# B&R Automation Studio project NAELD004C00R10L518F00 (part 31)

#### Local.var - Do Not Change!!!
```iecst
(*2019-06-17*)
(**)
(*Local Action, State & Status*)
VAR
	eAct : eConvAction := ConvActIdle;
	eStat : eConvAction := ConvActIdle;
	eStatus : eFBStatus := Idle;
	udiStatus : UDINT := 0;
	sStatTxt : STRING[200] := '';
	a_sStatText : ARRAY[0..60] OF STRING[200] := ['Idling','Initializing','Initializing With Reverse','Initializing With Pusher','Initializing With Puller','Initializing With Motorised Puller','Initializing With Reject','Initializing With Inspection','Entering Board','Entering Board Until Inlet Signal Off','Entering Board With Reverse','Reversing Board','Reversing Board With Immediate Start Conv','Entering Board With Puller','Entering Board With Reject','Entering Board With Inspection','Pre Exiting Board','Resuming Reject Board',2('Exiting Board'),2('Exiting Board With Pusher'),'Pusher Setting All Control','Pusher Resetting All Control','Pusher Setting Extend','Pusher Setting Retract','Pusher Extending','Pusher Retracting','Puller Setting All Control','Puller Resetting All Control','Puller Setting Extend','Puller Setting Retract','Puller Extending','Puller Retracting','Rotating Setting All Control','Rotating Resetting All Control','Rotating Setting Home','Rotating Setting Remote','Rotating Turning Home','Rotating Turning Remote','Reject Setting All Control','Reject Resetting All Control','Reject Setting Up','Reject Setting Down','Reject Going Up','Reject Going Down','Stopping','Stopping With Pusher','Stopping With Puller','Stopping With Reject','Turning On Motor Signal','Turning On Motor Direction','Turning Off Motor Signal','Turning Off Motor Direction','Turning On All Motor Output','Turning Off All Motor Output',5('')];
END_VAR
(**)
(*Local Alarm*)
VAR
	tyAlmData : tyAlmDat;
	a_tyAlmText : ARRAY[10000..10199] OF tyAlmTxt := [(sAlmText:='Multi Board Detected While Conveyor Initial',sRcyText:='Operation Interrupted By Multiple Board. Remove Extra Boards And Resume Operation.'),(sAlmText:='Board Not Present At Outlet Sensor (L - R) While Conveyor Initial',sRcyText:='Operation Interrupted By Jam Board. Remove The Jam Board To Resume Operation.'),(sAlmText:='Board Not Present At Outlet Sensor (R - L) While Conveyor Initial',sRcyText:='Operation Interrupted By Jam Board. Remove The Jam Board To Resume Operation.'),(sAlmText:='Multi Board Detected While Conveyor Initial With Reverse',sRcyText:='Operation Interrupted By Multiple Board. Remove Extra Boards And Resume Operation.'),(sAlmText:='Board Not Present At Outlet Sensor (L - R) While Conveyor Initial With Reverse',sRcyText:='Operation Interrupted By Jam Board. Remove The Jam Board To Resume Operation.'),(sAlmText:='Board Not Present At Outlet Sensor (R - L) While Conveyor Initial With Reverse',sRcyText:='Operation Interrupted By Jam Board. Remove The Jam Board To Resume Operation.'),(sAlmText:='Pusher Extend Sensor Off Time Out In Retract Check While Conveyor Initial With Pusher',sRcyText:='Sensor Timeout Expired Before Operation Completed. Sensor Operation Is Abnormal. Solve The Error To Resume Operation.'),(sAlmText:='Pusher Retract Sensor On Time Out In Retract Check While Conveyor Initial With Pusher',sRcyText:='Sensor Timeout Expired Before Operation Completed. Sensor Operation Is Abnormal. Solve The Error To Resume Operation.'),(sAlmText:='Pusher Retract Safety Sensor Error In Retract Check While Conveyor Initial With Pusher',sRcyText:='Safety System Has Been Triggered. All Operations Are Disable. Remove the Obstacle That Triggered The Safety Interlock To Resume Operation.'),(sAlmText:='Multi Board Detected While Conveyor Initial With Pusher',sRcyText:='Operation Interrupted By Multiple Board. Remove Extra Boards And Resume Operation.'),(sAlmText:='Board Not Present At Outlet Sensor (L - R) While Conveyor Initial With Pusher',sRcyText:='Operation Interrupted By Jam Board. Remove The Jam Board To Resume Operation.'),(sAlmText:='Board Not Present At Outlet Sensor (R - L) While Conveyor Initial With Pusher',sRcyText:='Operation Interrupted By Jam Board. Remove The Jam Board To Resume Operation.'),(sAlmText:='Rotator Home Sensor On Time Out In Home Check While Conveyor Initial With Puller',sRcyText:='Sensor Timeout Expired Before Operation Completed. Sensor Operation Is Abnormal. Solve The Error To Resume Operation.'),(sAlmText:='Rotator Remote Sensor Off Time Out In Home Check While Conveyor Initial With Puller',sRcyText:='Sensor Timeout Expired Before Operation Completed. Sensor Operation Is Abnormal. Solve The Error To Resume Operation.'),(sAlmText:='Rotator Home Safety Sensor Error In Home Check While Conveyor Initial With Puller',sRcyText:='Safety System Has Been Triggered. All Operations Are Disable. Remove the Obstacle That Triggered The Safety Interlock To Resume Operation.'),(sAlmText:='Puller Extend Sensor Off Time Out In Retract Check While Conveyor Initial With Puller',sRcyText:='Sensor Timeout Expired Before Operation Completed. Sensor Operation Is Abnormal. Solve The Error To Resume Operation.'),(sAlmText:='Puller Retract Sensor On Time Out In Retract Check While Conveyor Initial With Puller',sRcyText:='Sensor Timeout Expired Before Operation Completed. Sensor Operation Is Abnormal. Solve The Error To Resume Operation.'),(sAlmText:='Puller Retract Safety Sensor Error In Retract Check While Conveyor Initial With Puller',sRcyText:='Safety System Has Been Triggered. All Operations Are Disable. Remove the Obstacle That Triggered The Safety Interlock To Resume Operation.'),(sAlmText:='Multi Board Detected While Conveyor Initial With Puller',sRcyText:='Operation Interrupted By Multiple Board. Remove Extra Boards And Resume Operation.'),(sAlmText:='Board Not Present At Outlet Sensor (L - R) While Conveyor Initial With Puller',sRcyText:='Operation Interrupted By Jam Board. Remove The Jam Board To Resume Operation.'),(sAlmText:='Board Not Present At Outlet Sensor (R - L) While Conveyor Initial With Puller',sRcyText:='Operation Interrupted By Jam Board. Remove The Jam Board To Resume Operation.'),(sAlmText:='Multi Board Detected While Conveyor Enter Board',sRcyText:='Operation Interrupted By Multiple Board. Remove Extra Boards And Resume Operation.'),(sAlmText:='Multi Board Detected While Conveyor Enter Board With Reverse',sRcyText:='Operation Interrupted By Multiple Board. Remove Extra Boards And Resume Operation.'),(sAlmText:='Puller Extend Sensor On Time Out In Extend Check While Conveyor Enter With Puller',sRcyText:='Sensor Timeout Expired Before Operation Completed. Sensor Operation Is Abnormal. Solve The Error To Resume Operation.'),(sAlmText:='Puller Retract Sensor Off Time Out In Extend Check While Conveyor Enter With Puller',sRcyText:='Sensor Timeout Expired Before Operation Completed. Sensor Operation Is Abnormal. Solve The Error To Resume Operation.'),(sAlmText:='Puller Extend Safety Sensor Error In Extend Check While Conveyor Enter With Puller',sRcyText:='Safety System Has Been Triggered. All Operations Are Disable. Remove the Obstacle That Triggered The Safety Interlock To Resume Operation.'),(sAlmText:='Rotator Home Sensor Off Time Out In Remote Check While Conveyor Enter With Puller',sRcyText:='Sensor Timeout Expired Before Operation Completed. Sensor Operation Is Abnormal. Solve The Error To Resume Operation.'),(sAlmText:='Rotator Remote Sensor On Time Out In Remote Check While Conveyor Enter With Puller',sRcyText:='Sensor Timeout Expired Before Operation Completed. Sensor Operation Is Abnormal. Solve The Error To Resume Operation.'),(sAlmText:='Rotator Remote Safety Sensor Error In Remote Check While Conveyor Enter With Puller',sRcyText:='Safety System Has Been Triggered. All Operations Are Disable. Remove the Obstacle That Triggered The Safety Interlock To Resume Operation.'),(sAlmText:='Puller Extend Sensor Off Time Out In Retract Check While Conveyor Enter With Puller',sRcyText:='Sensor Timeout Expired Before Operation Completed. Sensor Operation Is Abnormal. Solve The Error To Resume Operation.'),(sAlmText:='Puller Retract Sensor On Time Out In Retract Check While Conveyor Enter With Puller',sRcyText:='Sensor Timeout Expired Before Operation Completed. Sensor Operation Is Abnormal. Solve The Error To Resume Operation.'),(sAlmText:='Puller Retract Safety Sensor Error In Retract Check While Conveyor Enter With Puller',sRcyText:='Safety System Has Been Triggered. All Operations Are Disable. Remove the Obstacle That Triggered The Safety Interlock To Resume Operation.'),(sAlmText:='Rotator Home Sensor On Time Out In Home Check While Conveyor Enter With Puller',sRcyText:='Sensor Timeout Expired Before Operation Completed. Sensor Operation Is Abnormal. Solve The Error To Resume Operation.'),(sAlmText:='Rotator Remote Sensor Off Time Out In Home Check While Conveyor Enter With Puller',sRcyText:='Sensor Timeout Expired Before Operation Completed. Sensor Operation Is Abnormal. Solve The Error To Resume Operation.'),(sAlmText:='Rotator Home Safety Sensor Error In Home Check While Conveyor Enter With Puller',sRcyText:='Safety System Has Been Triggered. All Operations Are Disable. Remove the Obstacle That Triggered The Safety Interlock To Resume Operation.'),(sAlmText:='Multi Board Detected While Conveyor Enter With Puller',sRcyText:='Operation Interrupted By Multiple Board. Remove Extra Boards And Resume Operation.'),(sAlmText:='Multi Board Detected While Conveyor Pre-Exit Board',sRcyText:='Operation Interrupted By Multiple Board. Remove Extra Boards And Resume Operation.'),(sAlmText:='Board Missing While Conveyor Pre-Exit Board',sRcyText:='Operation Interrupted By Jam Board. Remove The Jam Board To Resume Operation.'),(sAlmText:='Multi Board Detected While Conveyor Exit Board',sRcyText:='Operation Interrupted By Multiple Board. Remove Extra Boards And Resume Operation.'),(sAlmText:='Multi Board Detected While Conveyor Exit Board With Pusher',sRcyText:='Operation Interrupted By Multiple Board. Remove Extra Boards And Resume Operation.'),(sAlmText:='Pusher Extend Sensor On Time Out In Extend Check While Conveyor Exit Board With Pusher',sRcyText:='Sensor Timeout Expired Before Operation Completed. Sensor Operation Is Abnormal. Solve The Error To Resume Operation.'),(sAlmText:='Pusher Retract Sensor Off Time Out In Extend Check While Conveyor Exit Board With Pusher',sRcyText:='Sensor Timeout Expired Before Operation Completed. Sensor Operation Is Abnormal. Solve The Error To Resume Operation.'),(sAlmText:='Pusher Extend Safety Sensor Error In Extend Check While Conveyor Exit Board With Pusher',sRcyText:='Safety System Has Been Triggered. All Operations Are Disable. Remove the Obstacle That Triggered The Safety Interlock To Resume Operation.'),(sAlmText:='Pusher Extend Sensor Off Time Out In Retract Check While Conveyor Exit Board With Pusher',sRcyText:='Sensor Timeout Expired Before Operation Completed. Sensor Operation Is Abnormal.Solve The Error To Resume Operation.'),(sAlmText:='Pusher Retract Sensor On Timeout In Retract Check While Conveyor Exit Board With Pusher',sRcyText:='Sensor Timeout Expired Before Operation Completed. Sensor Operation Is Abnormal. Solve The Error To Resume Operation.'),(sAlmText:='Pusher Retract Safety Sensor Error In Retract Check While Conveyor Exit Board With Pusher',sRcyText:='Safety System Has Been Triggered. All Operations Are Disable. Remove the Obstacle That Triggered The Safety Interlock To Resume Operation.'),(sAlmText:='Pusher Extend Sensor On Time Out In Extend Check While Pusher Extend',sRcyText:='Sensor Timeout Expired Before Operation Completed. Sensor Operation Is Abnormal. Solve The Error To Resume Operation.'),(sAlmText:='Pusher Retract Sensor Off Time Out In Extend Check While Pusher Extend',sRcyText:='Sensor Timeout Expired Before Operation Completed. Sensor Operation Is Abnormal. Solve The Error To Resume Operation.'),(sAlmText:='Pusher Extend Safety Sensor Error In Extend Check While Pusher Extend',sRcyText:='Safety System Has Been Triggered. All Operations Are Disable. Remove the Obstacle That Triggered The Safety Interlock To Resume Operation.'),(sAlmText:='Pusher Extend Sensor Off Time Out In Retract Check While Pusher Retract',sRcyText:='Sensor Timeout Expired Before Operation Completed. Sensor Operation Is Abnormal. Solve The Error To Resume Operation.'),(sAlmText:='Pusher Retract Sensor On Time Out In Retract Check While Pusher Retract',sRcyText:='Sensor Timeout Expired Before Operation Completed. Sensor Operation Is Abnormal. Solve The Error To Resume Operation.'),(sAlmText:='Pusher Retract Safety Sensor Error In Retract Check While Pusher Retract',sRcyText:='Safety System Has Been Triggered. All Operations Are Disable. Remove the Obstacle That Triggered The Safety Interlock To Resume Operation.'),(sAlmText:='Puller Extend Sensor On Time Out In Extend Check While Puller Extend',sRcyText:='Sensor Timeout Expired Before Operation Completed. Sensor Operation Is Abnormal. Solve The Error To Resume Operation.'),(sAlmText:='Puller Retract Sensor Off Time Out In Extend Check While Puller Extend',sRcyText:='Sensor Timeout Expired Before Operation Completed. Sensor Operation Is Abnormal. Solve The Error To Resume Operation.'),(sAlmText:='Puller Extend Safety Sensor Error In Extend Check While Puller Extend',sRcyText:='Safety System Has Been Triggered. All Operations Are Disable. Remove the Obstacle That Triggered The Safety Interlock To Resume Operation.'),(sAlmText:='Puller Extend Sensor Off Time Out In Retract Check While Puller Retract',sRcyText:='Sensor Timeout Expired Before Operation Completed. Sensor Operation Is Abnormal. Solve The Error To Resume Operation.'),(sAlmText:='Puller Retract Sensor On Time Out In Retract Check While Puller Retract',sRcyText:='Sensor Timeout Expired Before Operation Completed. Sensor Operation Is Abnormal. Solve The Error To Resume Operation.'),(sAlmText:='Puller Retract Safety Sensor Error In Retract Check While Puller Retract',sRcyText:='Safety System Has Been Triggered. All Operations Are Disable. Remove the Obstacle That Triggered The Safety Interlock To Resume Operation.'),(sAlmText:='Rotator Home Sensor On Time Out In Home Check While Rotator Home',sRcyText:='Sensor Timeout Expired Before Operation Completed. Sensor Operation Is Abnormal. Solve The Error To Resume Operation.'),(sAlmText:='Rotator Remote Sensor Off Time Out In Home Check While Rotator Home',sRcyText:='Sensor Timeout Expired Before Operation Completed. Sensor Operation Is Abnormal. Solve The Error To Resume Operation.'),(sAlmText:='Rotator Home Safety Sensor Error In Home Check While Rotator Home',sRcyText:='Safety System Has Been Triggered. All Operations Are Disable. Remove the Obstacle That Triggered The Safety Interlock To Resume Operation.'),(sAlmText:='Rotator Home Sensor Off Time Out In Remote Check While Rotator Remote',sRcyText:='Sensor Timeout Expired Before Operation Completed. Sensor Operation Is Abnormal. Solve The Error To Resume Operation.'),(sAlmText:='Rotator Remote Sensor On Time Out In Remote Check While Rotator Remote',sRcyText:='Sensor Timeout Expired Before Operation Completed. Sensor Operation Is Abnormal. Solve The Error To Resume Operation.'),(sAlmText:='Rotator Remote Safety Sensor Error In Remote Check While Rotator Remote',sRcyText:='Safety System Has Been Triggered. All Operations Are Disable. Remove the Obstacle That Triggered The Safety Interlock To Resume Operation.'),(sAlmText:='Pusher Extend Sensor Off Time Out In Retract Check While Stop With Pusher',sRcyText:='Sensor Timeout Expired Before Operation Completed. Sensor Operation Is Abnormal. Solve The Error To Resume Operation.'),(sAlmText:='Pusher Retract Sensor On Time Out In Retract Check While Stop With Pusher',sRcyText:='Sensor Timeout Expired Before Operation Completed. Sensor Operation Is Abnormal. Solve The Error To Resume Operation.'),(sAlmText:='Pusher Retract Safety Sensor Error In Retract Check While Stop With Pusher',sRcyText:='Safety System Has Been Triggered. All Operations Are Disable. Remove the Obstacle That Triggered The Safety Interlock To Resume Operation.'),(sAlmText:='Rotator Home Sensor On Time Out In Home Check While Stop With Puller',sRcyText:='Sensor Timeout Expired Before Operation Completed. Sensor Operation Is Abnormal. Solve The Error To Resume Operation.'),(sAlmText:='Rotator Remote Sensor Off Time Out In Home Check While Stop With Puller',sRcyText:='Sensor Timeout Expired Before Operation Completed. Sensor Operation Is Abnormal. Solve The Error To Resume Operation.'),(sAlmText:='Rotator Home Safety Sensor Error In Home Check While Stop With Puller',sRcyText:='Safety System Has Been Triggered. All Operations Are Disable. Remove the Obstacle That Triggered The Safety Interlock To Resume Operation.'),(sAlmText:='Puller Extend Sensor Off Time Out In Retract Check While Stop With Puller',sRcyText:='Sensor Timeout Expired Before Operation Completed. Sensor Operation Is Abnormal. Solve The Error To Resume Operation.'),(sAlmText:='Puller Retract Sensor On Time Out In Retract Check While Stop With Puller',sRcyText:='Sensor Timeout Expired Before Operation Completed. Sensor Operation Is Abnormal. Solve The Error To Resume Operation.'),(sAlmText:='Puller Retract Safety Sensor Error In Retract Check While Stop With Puller',sRcyText:='Safety System Has Been Triggered. All Operations Are Disable. Remove the Obstacle That Triggered The Safety Interlock To Resume Operation.'),(sAlmText:='Reject Up Sensor On Time Out In Up Check While Reject Up',sRcyText:='Sensor Timeout Expired Before Operation Completed. Sensor Operation Is Abnormal. Solve The Error To Resume Operation.'),(sAlmText:='Reject Down Sensor Off Time Out In Up Check While Reject Up',sRcyText:='Sensor Timeout Expired Before Operation Completed. Sensor Operation Is Abnormal. Solve The Error To Resume Operation.'),(sAlmText:='Reject Up Safety Sensor Error In Up Check While Reject Up',sRcyText:='Safety System Has Been Triggered. All Operations Are Disable. Remove the Obstacle That Triggered The Safety Interlock To Resume Operation.'),(sAlmText:='Reject Up Sensor Off Time Out In Down Check While Reject Down',sRcyText:='Sensor Timeout Expired Before Operation Completed. Sensor Operation Is Abnormal. Solve The Error To Resume Operation.'),(sAlmText:='Reject Down Sensor On Time Out In Down Check While Reject Down',sRcyText:='Sensor Timeout Expired Before Operation Completed. Sensor Operation Is Abnormal. Solve The Error To Resume Operation.'),(sAlmText:='Reject Down Safety Sensor Error In Down Check While Reject Down',sRcyText:='Safety System Has Been Triggered. All Operations Are Disable. Remove the Obstacle That Triggered The Safety Interlock To Resume Operation.'),(sAlmText:='Multi Board Detected While Conveyor Initial With Reject',sRcyText:='Operation Interrupted By Multiple Board. Remove Extra Boards And Resume Operation.'),(sAlmText:='Board Not Present At Outlet Or Middle Sensor (L - R) While Conveyor Initial With Reject',sRcyText:='Operation Interrupted By Jam Board. Remove The Jam Board To Resume Operation.'),(sAlmText:='Board Not Present At Outlet Or Middle Sensor (R - L) While Conveyor Initial With Reject',sRcyText:='Operation Interrupted By Jam Board. Remove The Jam Board To Resume Operation.'),(sAlmText:='Reject Up Sensor On Time Out In Up Check While Conveyor Initial With Reject',sRcyText:='Sensor Timeout Expired Before Operation Completed. Sensor Operation Is Abnormal. Solve The Error To Resume Operation.'),(sAlmText:='Reject Down Sensor Off Time Out In Up Check While Conveyor Initial With Reject',sRcyText:='Sensor Timeout Expired Before Operation Completed. Sensor Operation Is Abnormal. Solve The Error To Resume Operation.'),(sAlmText:='Reject Up Safety Sensor Error In Up Check While Conveyor Initial With Reject',sRcyText:='Safety System Has Been Triggered. All Operations Are Disable. Remove the Obstacle That Triggered The Safety Interlock To Resume Operation.'),(sAlmText:='Multi Board Detected While Conveyor Initial With Inspect',sRcyText:='Operation Interrupted By Multiple Board. Remove Extra Boards And Resume Operation.'),(sAlmText:='Board Not Present At Outlet Or Middle Sensor (L - R) While Conveyor Initial With Inspection',sRcyText:='Operation Interrupted By Jam Board. Remove The Jam Board To Resume Operation.'),(sAlmText:='Board Not Present At Outlet Or Middle Sensor (R - L) While Conveyor Initial With Inspection',sRcyText:='Operation Interrupted By Jam Board. Remove The Jam Board To Resume Operation.'),(sAlmText:='Reject Up Sensor On Time Out In Up Check While Conveyor Initial With Reject',sRcyText:='Sensor Timeout Expired Before Operation Completed. Sensor Operation Is Abnormal. Solve The Error To Resume Operation.'),(sAlmText:='Reject Down Sensor Off Time Out In Up Check While Conveyor Initial With Reject',sRcyText:='Sensor Timeout Expired Before Operation Completed. Sensor Operation Is Abnormal. Solve The Error To Resume Operation.'),(sAlmText:='Reject Up Safety Sensor Error In Up Check While Conveyor Initial With Reject',sRcyText:='Safety System Has Been Triggered. All Operations Are Disable. Remove the Obstacle That Triggered The Safety Interlock To Resume Operation.'),(sAlmText:='Multi Board Detected While Conveyor Initial With Reject',sRcyText:='Operation Interrupted By Multiple Board. Remove Extra Boards And Resume Operation.'),(sAlmText:='Board Not Present At Outlet Sensor (L - R) While Conveyor Initial With Reject',sRcyText:='Operation Interrupted By Jam Board. Remove The Jam Board To Resume Operation.'),(sAlmText:='Board Not Present At Outlet Sensor (R - L) While Conveyor Initial With Reject',sRcyText:='Operation Interrupted By Jam Board. Remove The Jam Board To Resume Operation.'),(sAlmText:='Multi Board Detected While Conveyor Entering With Reject',sRcyText:='Operation Interrupted By Multiple Board. Remove Extra Boards And Resume Operation.'),(sAlmText:='Reject Up Sensor On Time Out In Up Check While Conveyor Entering With Reject',sRcyText:='Sensor Timeout Expired Before Operation Completed. Sensor Operation Is Abnormal. Solve The Error To Resume Operation.'),(sAlmText:='Reject Down Sensor Off Time Out In Up Check While Conveyor Entering With Reject',sRcyText:='Sensor Timeout Expired Before Operation Completed. Sensor Operation Is Abnormal. Solve The Error To Resume Operation.'),(sAlmText:='Reject Up Safety Sensor Error In Up Check While Conveyor Entering With Reject',sRcyText:='Safety System Has Been Triggered. All Operations Are Disable. Remove the Obstacle That Triggered The Safety Interlock To Resume Operation.'),(sAlmText:='Multi Board Detected While Conveyor Entering With Inspection',sRcyText:='Operation Interrupted By Multiple Board. Remove Extra Boards And Resume Operation.'),(sAlmText:='Board Detect In Middle Sensor While Resuming Rejected Board',sRcyText:='Operation Interrupted By Jam Board. Remove The Jam Board To Resume Operation.'),(sAlmText:='Reject Up Sensor Off Time Out In Down Check While Resuming Rejected Board',sRcyText:='Sensor Timeout Expired Before Operation Completed. Sensor Operation Is Abnormal. Solve The Error To Resume Operation.'),(sAlmText:='Reject Down Sensor On Time Out In Down Check While Resuming Rejected Board',sRcyText:='Sensor Timeout Expired Before Operation Completed. Sensor Operation Is Abnormal. Solve The Error To Resume Operation.'),(sAlmText:='Reject Down Safety Sensor Error In Down Check While Resuming Rejected Board',sRcyText:='Safety System Has Been Triggered. All Operations Are Disable. Remove the Obstacle That Triggered The Safety Interlock To Resume Operation.'),(sAlmText:='Multi Board Detected While Resuming Rejected Board',sRcyText:='Operation Interrupted By Multiple Board. Remove Extra Boards And Resume Operation.'),(sAlmText:='Board Not Present At Outlet Sensor (L - R) While Resuming Rejected Board',sRcyText:='Operation Interrupted By Jam Board. Remove The Jam Board To Resume Operation.'),(sAlmText:='Board Not Present At Outlet Sensor (R - L) While Resuming Rejected Board',sRcyText:='Operation Interrupted By Jam Board. Remove The Jam Board To Resume Operation.'),(sAlmText:='Multi Board Detected While Conveyor Exit Board',sRcyText:='Operation Interrupted By Multiple Board. Remove Extra Boards And Resume Operation.'),(sAlmText:='Multi Board Detected While Conveyor Exit Board With Pusher',sRcyText:='Operation Interrupted By Multiple Board. Remove Extra Boards And Resume Operation.'),(sAlmText:='Pusher Extend Sensor On Time Out In Extend Check While Conveyor Exit Board With Pusher',sRcyText:='Sensor Timeout Expired Before Operation Completed. Sensor Operation Is Abnormal. Solve The Error To Resume Operation.'),(sAlmText:='Pusher Retract Sensor Off Time Out In Extend Check While Conveyor Exit Board With Pusher',sRcyText:='Sensor Timeout Expired Before Operation Completed. Sensor Operation Is Abnormal. Solve The Error To Resume Operation.'),(sAlmText:='Pusher Extend Safety Sensor Error In Extend Check While Conveyor Exit Board With Pusher',sRcyText:='Safety System Has Been Triggered. All Operations Are Disable. Remove the Obstacle That Triggered The Safety Interlock To Resume Operation.'),(sAlmText:='Pusher Extend Sensor Off Time Out In Retract Check While Conveyor Exit Board With Pusher',sRcyText:='Sensor Timeout Expired Before Operation Completed. Sensor Operation Is Abnormal. Solve The Error To Resume Operation.'),(sAlmText:='Pusher Retract Sensor On Time Out In Retract Check While Conveyor Exit Board With Pusher',sRcyText:='Sensor Timeout Expired Before Operation Completed. Sensor Operation Is Abnormal. Solve The Error To Resume Operation.'),(sAlmText:='Pusher Retract Safety Sensor Error In Retract Check While Conveyor Exit Board With Pusher',sRcyText:='Safety System Has Been Triggered. All Operations Are Disable. Remove the Obstacle That Triggered The Safety Interlock To Resume Operation.'),(sAlmText:='Transfer In Time Out While Conveyor Enter Board',sRcyText:='Timeout Expired Before Operation Completed. Transmission Abnormal. Remove the Obstacle (If Exists) To Resume Operation.'),(sAlmText:='Transfer In Time Out While Conveyor Enter Board With Reverse',sRcyText:='Timeout Expired Before Operation Completed. Transmission Abnormal. Remove the Obstacle (If Exists) To Resume Operation.'),(sAlmText:='Transfer In Time Out While Conveyor Enter With Puller',sRcyText:='Timeout Expired Before Operation Completed. Transmission Abnormal. Remove the Obstacle (If Exists) To Resume Operation.'),(sAlmText:='Transfer In Time Out While Conveyor Entering With Reject',sRcyText:='Timeout Expired Before Operation Completed. Transmission Abnormal. Remove the Obstacle (If Exists) To Resume Operation.'),(sAlmText:='Transfer In Time Out While Conveyor Entering With Inspection',sRcyText:='Timeout Expired Before Operation Completed. Transmission Abnormal. Remove the Obstacle (If Exists) To Resume Operation.'),(sAlmText:='Transfer Out Time Out While Conveyor Exit Board',sRcyText:='Timeout Expired Before Operation Completed. Transmission Abnormal. Remove the Obstacle (If Exists) To Resume Operation.'),(sAlmText:='Transfer Out Time Out While Conveyor Exit Board With Pusher',sRcyText:='Timeout Expired Before Operation Completed. Transmission Abnormal. Remove the Obstacle (If Exists) To Resume Operation.'),(sAlmText:='Transfer Out Time Out While Conveyor Exit Board',sRcyText:='Timeout Expired Before Operation Completed. Transmission Abnormal. Remove the Obstacle (If Exists) To Resume Operation.'),(sAlmText:='Transfer Out Time Out While Conveyor Exit Board With Pusher',sRcyText:='Timeout Expired Before Operation Completed. Transmission Abnormal. Remove the Obstacle (If Exists) To Resume Operation.'),(sAlmText:='Multi Board Detected While Conveyor Enter Board To Inlet Off',sRcyText:='Operation Interrupted By Multiple Board. Remove Extra Boards And Resume Operation.'),(sAlmText:='Transfer In Time Out While Conveyor Enter Board To Inlet Off',sRcyText:='Timeout Expired Before Operation Completed. Transmission Abnormal. Remove the Obstacle (If Exists) To Resume Operation.'),(sAlmText:='Puller AntiJam Sensor On',sRcyText:='Board Jam During Puller Is Retracting'),(0),0,72((0))];
END_VAR
(**)
(*Local Output*)
VAR
	bHvBrd : BOOL;
	bRejHvBrd : BOOL;
	bInspHvBrd : BOOL;
	bGdBrd : BOOL;
	bLmtSenActivated : BOOL;
	bMtrSigOnOrLToR : BOOL;
	bMtrDirOrRToL : BOOL;
	bPshrExtCtrl : BOOL;
	bPshrTwoOutputControl : BOOL := FALSE;
	bPshrExtended : BOOL;
	bPshrRetracted : BOOL;
	bPullerExtCtrl : BOOL;
	bPullerRetCtrl : BOOL;
	bPullerTwoOutputControl : BOOL := TRUE;
	bPullerExtended : BOOL;
	bPullerRetracted : BOOL;
	bRotRemoteCtrl : BOOL;
	bRotTwoOutputControl : BOOL := FALSE;
	bRotAtRemote : BOOL;
	bRotAtHome : BOOL;
	bRejectUpCtrl : BOOL;
	bRejectDownCtrl : BOOL;
	bRejectTwoOutputControl : BOOL := TRUE;
	bRejectAtUp : BOOL;
	bRejectAtDown : BOOL;
END_VAR
(**)
(*Local Input*)
VAR
	udiRstErr : UDINT := 0;
	bPrep : BOOL := TRUE;
	bEn : BOOL := TRUE;
	bDis : BOOL := FALSE;
	bManual : BOOL := FALSE;
	bLongBrdPrep : BOOL := FALSE;
	bLongBrdEn : BOOL := FALSE;
	bOnDirMod : BOOL := FALSE;
	diInitTm : DINT := 10000;
	diRevDlyTm : DINT := 500;
	tMtrOffDlyTm : TIME := T#0S;
	diTxInTimeOut : DINT := 10000;
	diTxOutTimeOut : DINT := 10000;
	eDirection : eConvDir := ConvDirLToR;
	bGdBrdInit : BOOL := TRUE;
	bGdBrdEnt : BOOL := TRUE;
	bLeftSen : BOOL := FALSE;
	bRightSen : BOOL := FALSE;
	bMiddleSen : BOOL := FALSE;
	bPullerChkSen : BOOL := FALSE;
	bPshrExtSen : BOOL := FALSE;
	bPshrRetSen : BOOL := FALSE;
	bPshrExtSafetySen : BOOL := TRUE;
	bPshrRetSafetySen : BOOL := TRUE;
	bPullerExtSen : BOOL := FALSE;
	bPullerRetSen : BOOL := FALSE;
	bPullerExtSafetySen : BOOL := TRUE;
	bPullerRetSafetySen : BOOL := TRUE;
	bRotHomeSen : BOOL := FALSE;
	bRotRemoteSen : BOOL := FALSE;
	bRotHomeSafetySen : BOOL := TRUE;
	bRotRemoteSafetySen : BOOL := TRUE;
	bRejectUpSen : BOOL := FALSE;
	bRejectDownSen : BOOL := FALSE;
	bRejectUpSafetySen : BOOL := TRUE;
	bRejectDownSafetySen : BOOL := TRUE;
	sProgNm : STRING[15] := 'Conv';
	tPshrExtTO : TIME := T#20s;
	tPshrRetTO : TIME := T#20s;
	tPullerExtTO : TIME := T#20s;
	tPullerRetTO : TIME := T#20s;
	tRotHomeTO : TIME := T#20s;
	tRotRemoteTO : TIME := T#20s;
	tRejectUpTO : TIME := T#20s;
	tRejectDownTO : TIME := T#20s;
	bNtSettingsLoadDone : BOOL := TRUE;
END_VAR
(**)
(*Local*)
VAR
	bRstErr : BOOL;
	udiRstErrOld : UDINT;
	bInitDone : BOOL;
	bInitialDone : BOOL;
	usiStep : USINT;
	bInletOff : BOOL;
	fbWaitTm : TON := (PT:=T#1s);
	fbBoardOffTm : TON := (PT:=T#2s);
	eStatOld : eConvAction := ConvActIdle;
	fbInit : fbConvSenToSenTm;
	fbEnt : fbConvSenToSen;
	fbRev : fbConvSenToSenTm1;
	fbPreExit : fbConvSenToSenTm;
	fbExit : fbConvSenToSenOff;
	fbExit1 : fbConvSenToSenOff1;
	fbLongBrd : fbConvLongBrd;
	fbStop : fbConvMtrOff;
	fbPshrExtChk : fbPneuExtRetSenExtChk;
	fbPshrRetChk : fbPneuExtRetSenRetChk;
	fbPullerExtChk : fbPneuExtRetSenExtChk;
	fbPullerRetChk : fbPneuExtRetSenRetChk;
	fbRotHomeChk : fbPneuExtRetSenExtChk;
	fbRotRemoteChk : fbPneuExtRetSenRetChk;
	fbRejectUpChk : fbPneuExtRetSenExtChk;
	fbRejectDownChk : fbPneuExtRetSenRetChk;
	fbRightSenTm : TON := (PT:=T#1s);
	fbRightSenTmOff : TON := (PT:=T#1s);
	udiModuleNum : UDINT := 1501;
END_VAR
```

### MagConv2Clp.typ - Change By Project
```iecst
(*2019-10-30*)
(**)
(*Action*)

TYPE
	eMagConv2ClpAction :
		(
		MagConv2ClpActIdle,
		MagConv2ClpActInit,
		MagConv2ClpActInitStopClp,
		MagConv2ClpActInitClpStop,
		MagConv2ClpActEnt,
		MagConv2ClpActEntStopClp,
		MagConv2ClpActEntClpStop,
		MagConv2ClpActPreExit,
		MagConv2ClpActPreExitClpr,
		MagConv2ClpActExit,
		MagConv2ClpActExit1,
		MagConv2ClpActExitClpr,
		MagConv2ClpActExit1Clpr,
		MagConv2ClpActFixClprSetAll,
		MagConv2ClpActFixClprRstAll,
		MagConv2ClpActFixClprSetClamp,
		MagConv2ClpActFixClprSetUnclamp,
		MagConv2ClpActFixClprClamp,
		MagConv2ClpActFixClprUnclamp,
		MagConv2ClpActRmtClprSetAll,
		MagConv2ClpActRmtClprRstAll,
		MagConv2ClpActRmtClprSetClamp,
		MagConv2ClpActRmtClprSetUnclamp,
		MagConv2ClpActRmtClprClamp,
		MagConv2ClpActRmtClprUnclamp,
		MagConv2ClpActStop,
		MagConv2ClpActStopClpr,
		MagConv2ClpActSetMtrSigOnOrLToR,
		MagConv2ClpActSetMtrDirOrRToL,
		MagConv2ClpActRstMtrSigOnOrLToR,
		MagConv2ClpActRstMtrDirOrRToL,
		MagConv2ClpActSetMtrAll,
		MagConv2ClpActRstMtrAll
		);
END_TYPE

(**)
```

### Program Logical/MagConv/MagConv2Clp1 (IEC) - 1.00.0 - NtConv v5.00.0 , NtPneu v5.00.0

#### Act_InitGlobal.st
```iecst
(** 2019-10-30 **)
ACTION Act_InitGlobal:

	(* Always Change If Project Change *)

	//Pass Data To Link
	p_bLinkOpsRun ACCESS p_OpsRun;

	p_bLinkDISafetyRlySig ACCESS p_DISafetyRlySig;

	p_bLinkMagSmallSen ACCESS p_DIMagConvSmallMagSen1;
	p_bLinkMagLargeSen ACCESS p_DIMagConvLargeMagSen1;
	p_bLinkFixClprUnClampSen ACCESS p_DIMag1FixedUnclampRS;
	p_bWidthChkInterrupt ACCESS p_DICurtainSen;
	p_bLinkFixClprClampSen ACCESS ADR(bFixClprClampSen);//p_DIMag1FixedSideDetect;//p_DIMag1FixedClampRS; //initLocal at 1st
	p_bLinkDO ACCESS p_DO;
	p_bLinkMagOpsStepMagMtyExit ACCESS p_OpsMagConvLD1MagMtyExit;
	p_bLinkDIMagEntSen ACCESS p_DIMagConvEntSen1;

	p_bLinkNtParamMagModelAutoVerify ACCESS p_NtParamProjMagAutoVerifyPrep;
	p_bRmtClprUnclampSen ACCESS p_DIMag1RemoteUnclampRS;
	p_tyDISettings ACCESS p_NtParamDISettings;

	//Pass Data To Internal Use
	p_udiRstErr ACCESS p_RstErrReset;
	p_bPrep ACCESS p_NtParamProjMag1ConvPrep;
	p_bManual ACCESS p_UIMnlMod;
	p_bOnDirMod ACCESS p_NtParamMagConv1OnDirMod;
	p_diInitTm ACCESS p_McParamMag1ConvRunTmOut;
	p_tMtrOffDlyTm ACCESS p_NtParamMagConv1MtrOffDlyTm;
	p_diTxInTimeOut ACCESS p_McParamMag1ConvRunTmOut;
	p_diTxOutTimeOut ACCESS p_McParamMag1ConvRunTmOut;
	p_eDirection ACCESS p_NtParamProjMagConvDir;
	p_sProgNm ACCESS p_NtParamMagConv1ProgNm;
	p_tClprClampTO ACCESS p_NtParamMagConv1ClprClampTO;
	p_tClprUnclampTO ACCESS p_NtParamMagConv1ClprUnclampTO;
//	p_bLeftSen ACCESS p_DIMagConvEntSen1;
	p_bRightSen	ACCESS p_DIMagPresentSen1;

	p_bNtSettingsLoadDone ACCESS p_StartupNtSettingsLoadDone;

	(* Always Change If Project Change *)

END_ACTION
```

#### Act_Link.st
```iecst
(** 2019-10-30 **)
ACTION Act_Link:

	IF p_bLinkDISafetyRlySig = FALSE THEN
		bFixClprClampCtrl	:= FALSE;
		bRmtClprClampCtrl	:= FALSE;
	END_IF

	p_bFixClprUnclampSen :=  p_bLinkFixClprUnClampSen; //unclamp

	IF p_bLinkNtParamMagModelAutoVerify THEN
		fbSmallLargeSenDlyTm(IN:= p_bLinkMagSmallSen OR p_bLinkMagLargeSen);
		IF fbSmallLargeSenDlyTm.Q THEN
			p_bFixClprClampSen := TRUE;
		ELSE
			p_bFixClprClampSen := FALSE;
		END_IF
	ELSE
		p_bFixClprClampSen := p_bLinkFixClprClampSen;
	END_IF

	p_bRmtClprClampSen := p_bLinkDO.bMag1RemoteClampCtrl;
	p_bRmtClprUnclampSen := NOT p_bLinkDO.bMag1RemoteClampCtrl;
	//	p_tMtrOffDlyTm	:= T#200ms;

	IF p_bLinkMagOpsStepMagMtyExit THEN
		fbLeftSenDelayTm(IN:= TRUE, PT:=  T#5000ms);
		IF fbLeftSenDelayTm.Q THEN
			p_bLeftSen := p_bLinkDIMagEntSen;
		END_IF
	ELSE
		p_bLeftSen := p_bLinkDIMagEntSen;
		fbLeftSenDelayTm(IN:= FALSE);
	END_IF

	//Clamp Sensor chk time
	IF p_tyDISettings.diMag1FixedSideDetect >0 THEN //fix side sensor used

		IF eStat = MagConv2ClpActInitStopClp AND usiStep = 3 OR
			eStat = MagConv2ClpActEntStopClp AND usiStep = 1 OR
			eStat = MagConv2ClpActFixClprClamp OR eStat = MagConv2ClpActFixClprUnclamp THEN //during clamp
			fbClpExtChkTm(IN:=TRUE);

			IF fbClpExtChkTm.Q THEN
				fbClpExtChkTm(IN:=FALSE);
				p_bLinkFixClprClampSen ACCESS p_DIMag1FixedSideDetect;
			ELSE
				p_bLinkFixClprClampSen ACCESS ADR(bFixClprClampSen);
			END_IF
		ELSE
			fbClpExtChkTm(IN:=FALSE);
			p_bFixClprClampSen := FALSE;
		END_IF
	ELSE //standard 2 RS
		p_bLinkFixClprClampSen ACCESS p_DIMag1FixedClampRS;
	END_IF

END_ACTION
```

#### Act_LinkAction.st
```iecst
(** 2019-10-30 **)
ACTION Act_LinkAction:

	IF p_bLinkOpsRun = TRUE THEN
		p_eAct ACCESS p_OpsMagConvLD1MagConv2ClpAct;
	ELSIF p_bManual = TRUE THEN
		p_eAct ACCESS p_UIMagConv2Clp1Act;
	ELSE
		p_eAct ACCESS ADR(eAct);
	END_IF

END_ACTION
```

### Program Logical/MagConv/MagConv2Clp2 (IEC) - 1.00.0 - NtConv v5.00.0 , NtPneu v5.00.0

#### InputRef_Link.var
```iecst
(*2019-10-30*)
(**)
VAR
	p_bLinkOpsRun : REFERENCE TO BOOL;
END_VAR
(**)
VAR
	p_bLinkDISafetyRlySig : REFERENCE TO BOOL;
	p_bLinkMagSmallSen : REFERENCE TO BOOL;
	p_bLinkMagLargeSen : REFERENCE TO BOOL;
	p_bLinkFixClprUnClampSen : REFERENCE TO BOOL;
	p_bLinkFixClprClampSen : REFERENCE TO BOOL;
	p_bLinkMagOpsStepMagMtyExit : REFERENCE TO BOOL;
	p_bLinkDIMagEntSen : REFERENCE TO BOOL;
	p_bLinkDO : REFERENCE TO tyDigitalOutput;
	p_bLinkNtParamMagModelAutoVerify : REFERENCE TO BOOL;
	p_tyDISettings : REFERENCE TO tyDigitalInputSettings;
END_VAR
```

#### Act_InitGlobal.st
```iecst
(** 2019-10-30 **)
ACTION Act_InitGlobal:

	(* Always Change If Project Change *)

	//Pass Data To Link
	p_bLinkOpsRun ACCESS p_OpsRun;

	p_bLinkDISafetyRlySig ACCESS p_DISafetyRlySig;

	p_bLinkMagSmallSen ACCESS p_DIMagConvSmallMagSen2;
	p_bLinkMagLargeSen ACCESS p_DIMagConvLargeMagSen2;
	p_bLinkFixClprUnClampSen ACCESS p_DIMag2FixedUnclampRS;
	p_bWidthChkInterrupt ACCESS p_DICurtainSen;
	p_bLinkFixClprClampSen ACCESS ADR(bFixClprClampSen);//p_DIMag2FixedSideDetect;//p_DIMag2FixedClampRS;
	p_bLinkDO ACCESS p_DO;
	p_bLinkMagOpsStepMagMtyExit ACCESS p_OpsMagConvLD2MagMtyExit;
	p_bLinkDIMagEntSen ACCESS p_DIMagConvEntSen2;

	p_bLinkNtParamMagModelAutoVerify ACCESS p_NtParamProjMagAutoVerifyPrep;
	p_bRmtClprUnclampSen ACCESS p_DIMag2RemoteUnclampRS;
	p_tyDISettings ACCESS p_NtParamDISettings;

	//Pass Data To Internal Use
	p_udiRstErr ACCESS p_RstErrReset;
	p_bPrep ACCESS p_NtParamProjMag2ConvPrep;
	p_bManual ACCESS p_UIMnlMod;
	p_bOnDirMod ACCESS p_NtParamMagConv2OnDirMod;
	p_diInitTm ACCESS p_McParamMag2ConvRunTmOut;
	p_tMtrOffDlyTm ACCESS p_NtParamMagConv2MtrOffDlyTm;
	p_diTxInTimeOut ACCESS p_McParamMag2ConvRunTmOut;
	p_diTxOutTimeOut ACCESS p_McParamMag2ConvRunTmOut;
	p_eDirection ACCESS p_NtParamProjMagConvDir;
	p_sProgNm ACCESS p_NtParamMagConv2ProgNm;
	p_tClprClampTO ACCESS p_NtParamMagConv2ClprClampTO;
	p_tClprUnclampTO ACCESS p_NtParamMagConv2ClprUnclampTO;
//	p_bLeftSen ACCESS p_DIMagConvEntSen2;
	p_bRightSen	ACCESS p_DIMagPresentSen2;

	p_bNtSettingsLoadDone ACCESS p_StartupNtSettingsLoadDone;

	(* Always Change If Project Change *)

END_ACTION
```

#### Act_Link.st
```iecst
(** 2019-10-30 **)
ACTION Act_Link:

	IF p_bLinkDISafetyRlySig = FALSE THEN
		bFixClprClampCtrl	:= FALSE;
		bRmtClprClampCtrl	:= FALSE;
	END_IF

	p_bFixClprUnclampSen :=  p_bLinkFixClprUnClampSen;

	IF p_bLinkNtParamMagModelAutoVerify THEN
		fbSmallLargeSenDlyTm(IN:= p_bLinkMagSmallSen OR p_bLinkMagLargeSen);
		IF fbSmallLargeSenDlyTm.Q THEN
			p_bFixClprClampSen := TRUE;
		ELSE
			p_bFixClprClampSen := FALSE;
		END_IF
	ELSE
		p_bFixClprClampSen := p_bLinkFixClprClampSen;
	END_IF

	p_bRmtClprClampSen := p_bLinkDO.bMag2RemoteClampCtrl;
	p_bRmtClprUnclampSen := NOT p_bLinkDO.bMag2RemoteClampCtrl;
//	p_tMtrOffDlyTm	:= T#200ms;

	IF p_bLinkMagOpsStepMagMtyExit THEN
		fbLeftSenDelayTm(IN:= TRUE, PT:=  T#5000ms);
		IF fbLeftSenDelayTm.Q THEN
			p_bLeftSen := p_bLinkDIMagEntSen;
		END_IF
	ELSE
		p_bLeftSen := p_bLinkDIMagEntSen;
		fbLeftSenDelayTm(IN:= FALSE);
	END_IF

	//Clamp Sensor chk time
	IF p_tyDISettings.diMag2FixedSideDetect >0 THEN //fix side sensor used

		IF eStat = MagConv2ClpActInitStopClp AND usiStep = 3 OR
			eStat = MagConv2ClpActEntStopClp AND usiStep = 1 OR
			eStat = MagConv2ClpActFixClprClamp OR eStat = MagConv2ClpActFixClprUnclamp THEN //during clamp
			fbClpExtChkTm(IN:=TRUE);

			IF fbClpExtChkTm.Q THEN
				fbClpExtChkTm(IN:=FALSE);
				p_bLinkFixClprClampSen ACCESS p_DIMag2FixedSideDetect;
			ELSE
				p_bLinkFixClprClampSen ACCESS ADR(bFixClprClampSen);
			END_IF
		ELSE
			fbClpExtChkTm(IN:=FALSE);
			p_bFixClprClampSen := FALSE;
		END_IF
	ELSE //standard 2 RS
		p_bLinkFixClprClampSen ACCESS p_DIMag2FixedClampRS;
	END_IF

END_ACTION
```

#### Act_LinkAction.st
```iecst
(** 2019-10-30 **)
ACTION Act_LinkAction:

	IF p_bLinkOpsRun = TRUE THEN
		p_eAct ACCESS p_OpsMagConvLD2MagConv2ClpAct;
	ELSIF p_bManual = TRUE THEN
		p_eAct ACCESS p_UIMagConv2Clp2Act;
	ELSE
		p_eAct ACCESS ADR(eAct);
	END_IF

END_ACTION
```

### Program Logical/MagConv/MagConv2Clp3 (IEC, version 1.00.0) - 1.00.0 - NtConv v5.00.0 , NtPneu v5.00.0

#### Act_InitGlobal.st - Change By Project
```iecst
(** 2019-10-30 **)
ACTION Act_InitGlobal:

	(* Always Change If Project Change *)

	//Pass Data To Link
	p_bLinkOpsRun ACCESS p_OpsRun;

	p_bLinkDISafetyRlySig ACCESS p_DISafetyRlySig;

	p_bLinkMagSmallSen ACCESS p_DIMagConvSmallMagSen3;
	p_bLinkMagLargeSen ACCESS p_DIMagConvLargeMagSen3;
	p_bLinkFixClprUnClampSen ACCESS p_DIMag3FixedUnclampRS;
	p_bWidthChkInterrupt ACCESS p_DICurtainSen;
	p_bLinkFixClprClampSen ACCESS ADR(bFixClprClampSen);// p_DIMag3FixedSideDetect;//p_DIMag3FixedClampRS;
	p_bLinkDO ACCESS p_DO;
	p_bLinkMagOpsStepMagMtyExit ACCESS p_OpsMagConvLD3MagMtyExit;
	p_bLinkDIMagEntSen ACCESS p_DIMagConvEntSen3;

	p_bLinkNtParamMagModelAutoVerify ACCESS p_NtParamProjMagAutoVerifyPrep;
	p_bRmtClprUnclampSen ACCESS p_DIMag3RemoteUnclampRS;
	p_tyDISettings ACCESS p_NtParamDISettings;

	//Pass Data To Internal Use
	p_udiRstErr ACCESS p_RstErrReset;
	p_bPrep ACCESS p_NtParamProjMag3ConvPrep;
	p_bManual ACCESS p_UIMnlMod;
	p_bOnDirMod ACCESS p_NtParamMagConv3OnDirMod;
	p_diInitTm ACCESS p_McParamMag3ConvRunTmOut;
	p_tMtrOffDlyTm ACCESS p_NtParamMagConv3MtrOffDlyTm;
	p_diTxInTimeOut ACCESS p_McParamMag3ConvRunTmOut;
	p_diTxOutTimeOut ACCESS p_McParamMag3ConvRunTmOut;
	p_eDirection ACCESS p_NtParamProjMagConvDir;
	p_sProgNm ACCESS p_NtParamMagConv3ProgNm;
	p_tClprClampTO ACCESS p_NtParamMagConv3ClprClampTO;
	p_tClprUnclampTO ACCESS p_NtParamMagConv3ClprUnclampTO;
//	p_bLeftSen ACCESS p_DIMagConvEntSen3;
	p_bRightSen	ACCESS p_DIMagPresentSen3;

	p_bNtSettingsLoadDone ACCESS p_StartupNtSettingsLoadDone;

	(* Always Change If Project Change *)

END_ACTION
```

#### Act_LinkAction.st - Change By Project
```iecst
(** 2019-10-30 **)
ACTION Act_LinkAction:

	IF p_bLinkOpsRun = TRUE THEN
		p_eAct ACCESS p_OpsMagConvLD3MagConv2ClpAct;
	ELSIF p_bManual = TRUE THEN
		p_eAct ACCESS p_UIMagConv2Clp3Act;
	ELSE
		p_eAct ACCESS ADR(eAct);
	END_IF

END_ACTION
```

#### Act_Link.st - Change By Project
```iecst
(** 2019-10-30 **)
ACTION Act_Link:

	IF p_bLinkDISafetyRlySig = FALSE THEN
		bFixClprClampCtrl	:= FALSE;
		bRmtClprClampCtrl	:= FALSE;
	END_IF

	p_bFixClprUnclampSen :=  p_bLinkFixClprUnClampSen;

	IF p_bLinkNtParamMagModelAutoVerify THEN
		fbSmallLargeSenDlyTm(IN:= p_bLinkMagSmallSen OR p_bLinkMagLargeSen);
		IF fbSmallLargeSenDlyTm.Q THEN
			p_bFixClprClampSen := TRUE;
		ELSE
			p_bFixClprClampSen := FALSE;
		END_IF
	ELSE
		p_bFixClprClampSen := p_bLinkFixClprClampSen;
	END_IF

	p_bRmtClprClampSen := p_bLinkDO.bMag3RemoteClampCtrl;
	p_bRmtClprUnclampSen := NOT p_bLinkDO.bMag3RemoteClampCtrl;
//	p_tMtrOffDlyTm	:= T#200ms;

	IF p_bLinkMagOpsStepMagMtyExit THEN
		fbLeftSenDelayTm(IN:= TRUE, PT:= T#5000ms);
		IF fbLeftSenDelayTm.Q THEN
			p_bLeftSen := p_bLinkDIMagEntSen;
		END_IF
	ELSE
		p_bLeftSen := p_bLinkDIMagEntSen;
		fbLeftSenDelayTm(IN:= FALSE);
	END_IF

	//Clamp Sensor chk time
	IF p_tyDISettings.diMag3FixedSideDetect >0 THEN //fix side sensor used

		IF eStat = MagConv2ClpActInitStopClp AND usiStep = 3 OR
			eStat = MagConv2ClpActEntStopClp AND usiStep = 1 OR
			eStat = MagConv2ClpActFixClprClamp OR eStat = MagConv2ClpActFixClprUnclamp THEN //during clamp
			fbClpExtChkTm(IN:=TRUE);

			IF fbClpExtChkTm.Q THEN
				fbClpExtChkTm(IN:=FALSE);
				p_bLinkFixClprClampSen ACCESS p_DIMag3FixedSideDetect;
			ELSE
				p_bLinkFixClprClampSen ACCESS ADR(bFixClprClampSen);
			END_IF
		ELSE
			fbClpExtChkTm(IN:=FALSE);
			p_bFixClprClampSen := FALSE;
		END_IF
	ELSE //standard 2 RS
		p_bLinkFixClprClampSen ACCESS p_DIMag3FixedClampRS;
	END_IF

END_ACTION
```

#### Local.var - Do Not Change!!!
```iecst
(*2019-10-30*)
(**)
(*Local Action, State & Status*)
VAR
	eAct : eMagConv2ClpAction := MagConv2ClpActIdle;
	eStat : eMagConv2ClpAction := MagConv2ClpActIdle;
	eStatus : eFBStatus := Idle;
	udiStatus : UDINT := 0;
	sStatTxt : STRING[200] := '';
	a_sStatText : ARRAY[0..50] OF STRING[200] := ['Idling','Initializing','Initializing With Stop Then Clamper','Initializing With Clamper Then Stop','Entering Board','Entering Board With Stop Then Clamper','Entering Board With Clamper Then Stop','Pre-Exiting Board','Pre-Exiting Board With Clamper',2('Exiting Board'),2('Exiting Board With Clamper'),'Fix/Bottom Clamper Setting All Control','Fix/Bottom Clamper Resetting All Control','Fix/Bottom Clamper Setting Clamp','Fix/Bottom Clamper Setting Unclamp','Fix/Bottom Clamper Clamp','Fix/Bottom Clampler Unclamp','Remote/Top Clamper Setting All Control','Remote/Top Clamper Resetting All Control','Remote/Top Clamper Setting Clamp','Remote/Top Clamper Setting Unclamp','Remote/Top Clamper Clamp','Remote/Top Clampler Unclamp','Stopping','Stopping With Clamper','Turning On Motor Signal','Turning On Motor Direction','Turning Off Motor Signal','Turning Off Motor Direction','Turning On All Motor Output','Turning Off All Motor Output',18('')];
END_VAR
(**)
(*Local Alarm*)
VAR
	tyAlmData : tyAlmDat;
	a_tyAlmText : ARRAY[10000..10099] OF tyAlmTxt := [(sAlmText:='Magazine Detected But Not Present At Outlet Sensor (L - R) While Magazine Conveyor Initial',sRcyText:='Operation Interrupted By Undetected Magazine. Adjusting The Magazine Or Remove The Present Magazine To Resume Operation.'),(sAlmText:='Magazine Detected But Not Present At Outlet Sensor (R - L) While Magazine Conveyor Initial',sRcyText:='Operation Interrupted By Undetected Magazine. Adjusting The Magazine Or Remove The Present Magazine To Resume Operation.'),(sAlmText:='Clamper Clamp Sensor Off Time Out In Unclamp Check While Conveyor Initial With Clamper',sRcyText:='Sensor Timeout Expired Before Operation Completed. Sensor Operation Is Abnormal. Solve The Error To Resume Operation.'),(sAlmText:='Clamper Unclamp Sensor On Time Out In Unclamp Check While Conveyor Initial With Clamper',sRcyText:='Sensor Timeout Expired Before Operation Completed. Sensor Operation Is Abnormal. Solve The Error To Resume Operation.'),(sAlmText:='Clamper Unclamp Safety Sensor Error In Unclamp Check While Conveyor Initial With Clamper',sRcyText:='Safety System Has Been Triggered. All Operations Are Disable. Remove the Obstacle That Triggered The Safety Interlock To Resume Operation.'),(sAlmText:='Magazine Detected But Not Present At Outlet Sensor (L - R) While Conveyor Initial With Clamper',sRcyText:='Operation Interrupted By Undetected Magazine. Adjusting The Magazine Or Remove The Present Magazine To Resume Operation.'),(sAlmText:='Magazine Detected But Not Present At Outlet Sensor (R - L) While Conveyor Initial With Clamper',sRcyText:='Operation Interrupted By Undetected Magazine. Adjusting The Magazine Or Remove The Present Magazine To Resume Operation.'),(sAlmText:='Clamper Clamp Sensor On Time Out In Clamp Check While Conveyor Initial With Clamper',sRcyText:='Sensor Timeout Expired Before Operation Completed. Sensor Operation Is Abnormal. Solve The Error To Resume Operation.'),(sAlmText:='Clamper Unclamp Sensor Off Time Out In Clamp Check While Conveyor Initial With Clamper',sRcyText:='Sensor Timeout Expired Before Operation Completed. Sensor Operation Is Abnormal. Solve The Error To Resume Operation.'),(sAlmText:='Clamper Clamp Safety Sensor Error In Clamp Check While Conveyor Initial With Clamper',sRcyText:='Safety System Has Been Triggered. All Operations Are Disable. Remove the Obstacle That Triggered The Safety Interlock To Resume Operation.'),(sAlmText:='Clamper Clamp Sensor On Time Out In Clamp Check While Conveyor Enter With Clamper',sRcyText:='Sensor Timeout Expired Before Operation Completed. Sensor Operation Is Abnormal. Solve The Error To Resume Operation.'),(sAlmText:='Clamper Unclamp Sensor Off Time Out In Clamp Check While Conveyor Enter With Clamper',sRcyText:='Sensor Timeout Expired Before Operation Completed. Sensor Operation Is Abnormal. Solve The Error To Resume Operation.'),(sAlmText:='Clamper Clamp Safety Sensor Error In Clamp Check While Conveyor Enter With Clamper',sRcyText:='Safety System Has Been Triggered. All Operations Are Disable. Remove the Obstacle That Triggered The Safety Interlock To Resume Operation.'),(sAlmText:='Clamper Clamp Sensor Off Time Out In Unclamp Check While Conveyor Exit With Clamper',sRcyText:='Sensor Timeout Expired Before Operation Completed. Sensor Operation Is Abnormal. Solve The Error To Resume Operation.'),(sAlmText:='Clamper Unclamp Sensor On Time Out In Unclamp Check While Conveyor Exit With Clamper',sRcyText:='Sensor Timeout Expired Before Operation Completed. Sensor Operation Is Abnormal. Solve The Error To Resume Operation.'),(sAlmText:='Clamper Unclamp Safety Sensor Error In Unclamp Check While Conveyor Exit With Clamper',sRcyText:='Safety System Has Been Triggered. All Operations Are Disable. Remove the Obstacle That Triggered The Safety Interlock To Resume Operation.'),(sAlmText:='Clamper Clamp Sensor On Time Out In Clamp Check While Clamper Clamp',sRcyText:='Sensor Timeout Expired Before Operation Completed. Sensor Operation Is Abnormal. Solve The Error To Resume Operation.'),(sAlmText:='Clamper Unclamp Sensor Off Time Out In Clamp Check While Clamper Clamp',sRcyText:='Sensor Timeout Expired Before Operation Completed. Sensor Operation Is Abnormal. Solve The Error To Resume Operation.'),(sAlmText:='Clamper Clamp Safety Sensor Error In Clamp Check While Clamper Clamp',sRcyText:='Safety System Has Been Triggered. All Operations Are Disable. Remove the Obstacle That Triggered The Safety Interlock To Resume Operation.'),(sAlmText:='Clamper Clamp Sensor Off Time Out In Unclamp Check While Clamper Unclamp',sRcyText:='Sensor Timeout Expired Before Operation Completed. Sensor Operation Is Abnormal. Solve The Error To Resume Operation.'),(sAlmText:='Clamper Unclamp Sensor On Time Out In Unclamp Check While Clamper Unclamp',sRcyText:='Sensor Timeout Expired Before Operation Completed. Sensor Operation Is Abnormal. Solve The Error To Resume Operation.'),(sAlmText:='Clamper Unclamp Safety Sensor Error In Unclamp Check While Clamper Unclamp',sRcyText:='Safety System Has Been Triggered. All Operations Are Disable. Remove the Obstacle That Triggered The Safety Interlock To Resume Operation.'),(sAlmText:='Clamper Clamp Sensor Off Time Out In Unclamp Check While Stop With Clamper',sRcyText:='Sensor Timeout Expired Before Operation Completed. Sensor Operation Is Abnormal. Solve The Error To Resume Operation.'),(sAlmText:='Clamper Unclamp Sensor On Time Out In Unclamp Check While Stop With Clamper',sRcyText:='Sensor Timeout Expired Before Operation Completed. Sensor Operation Is Abnormal. Solve The Error To Resume Operation.'),(sAlmText:='Clamper Unclamp Safety Sensor Error In Unclamp Check While Stop With Clamper',sRcyText:='Safety System Has Been Triggered. All Operations Are Disable. Remove the Obstacle That Triggered The Safety Interlock To Resume Operation.'),(sAlmText:='Clamper Clamp Sensor Off Time Out In Unclamp Check While Conveyor Exit With Clamper',sRcyText:='Sensor Timeout Expired Before Operation Completed. Sensor Operation Is Abnormal. Solve The Error To Resume Operation.'),(sAlmText:='Clamper Unclamp Sensor On Time Out In Unclamp Check While Conveyor Exit With Clamper',sRcyText:='Sensor Timeout Expired Before Operation Completed. Sensor Operation Is Abnormal. Solve The Error To Resume Operation.'),(sAlmText:='Clamper Unclamp Safety Sensor Error In Unclamp Check While Conveyor Exit With Clamper',sRcyText:='Safety System Has Been Triggered. All Operations Are Disable. Remove the Obstacle That Triggered The Safety Interlock To Resume Operation.'),2((sAlmText:='Transfer In Time Out While Entering Magazine',sRcyText:='Timeout Expired Before Operation Completed. Transmission Abnormal. Remove the Obstacle (If Exists) To Resume Operation.')),(sAlmText:='Transfer Out Time Out While Exiting Magazine',sRcyText:='Timeout Expired Before Operation Completed. Transmission Abnormal. Remove the Obstacle (If Exists) To Resume Operation.'),(sAlmText:='Transfer Out Time Out While Conveyor Exit With Clamper',sRcyText:='Timeout Expired Before Operation Completed. Transmission Abnormal. Remove the Obstacle (If Exists) To Resume Operation.'),(sAlmText:='Transfer Out Time Out While Exiting Magazine',sRcyText:='Timeout Expired Before Operation Completed. Transmission Abnormal. Remove the Obstacle (If Exists) To Resume Operation.'),(sAlmText:='Transfer Out Time Out While Conveyor Exit With Clamper',sRcyText:='Timeout Expired Before Operation Completed. Transmission Abnormal. Remove the Obstacle (If Exists) To Resume Operation.'),(sAlmText:='Clamper Clamp Sensor On Time Out In Clamp Check While Conveyor Enter With Clamper',sRcyText:='Sensor Timeout Expired Before Operation Completed. Sensor Operation Is Abnormal. Solve The Error To Resume Operation.'),(sAlmText:='Clamper Unclamp Sensor Off Time Out In Clamp Check While Conveyor Enter With Clamper',sRcyText:='Sensor Timeout Expired Before Operation Completed. Sensor Operation Is Abnormal. Solve The Error To Resume Operation.'),(sAlmText:='Clamper Clamp Safety Sensor Error In Clamp Check While Conveyor Enter With Clamper',sRcyText:='Safety System Has Been Triggered. All Operations Are Disable. Remove the Obstacle That Triggered The Safety Interlock To Resume Operation.'),(sAlmText:='Transfer In Time Out While Entering Magazine',sRcyText:='Timeout Expired Before Operation Completed. Transmission Abnormal. Remove the Obstacle (If Exists) To Resume Operation.'),(sAlmText:='Clamper Clamp Sensor Off Time Out In Unclamp Check While Conveyor Initial With Clamper',sRcyText:='Sensor Timeout Expired Before Operation Completed. Sensor Operation Is Abnormal. Solve The Error To Resume Operation.'),(sAlmText:='Clamper Unclamp Sensor On Time Out In Unclamp Check While Conveyor Initial With Clamper',sRcyText:='Sensor Timeout Expired Before Operation Completed. Sensor Operation Is Abnormal. Solve The Error To Resume Operation.'),(sAlmText:='Clamper Unclamp Safety Sensor Error In Unclamp Check While Conveyor Initial With Clamper',sRcyText:='Safety System Has Been Triggered. All Operations Are Disable. Remove the Obstacle That Triggered The Safety Interlock To Resume Operation.'),(sAlmText:='Magazine Detected But Not Present At Outlet Sensor (L - R) While Conveyor Initial With Clamper',sRcyText:='Operation Interrupted By Undetected Magazine. Adjusting The Magazine Or Remove The Present Magazine To Resume Operation.'),(sAlmText:='Magazine Detected But Not Present At Outlet Sensor (R - L) While Conveyor Initial With Clamper',sRcyText:='Operation Interrupted By Undetected Magazine. Adjusting The Magazine Or Remove The Present Magazine To Resume Operation.'),(sAlmText:='Clamper Clamp Sensor On Time Out In Clamp Check While Conveyor Initial With Clamper',sRcyText:='Sensor Timeout Expired Before Operation Completed. Sensor Operation Is Abnormal. Solve The Error To Resume Operation.'),(sAlmText:='Clamper Unclamp Sensor Off Time Out In Clamp Check While Conveyor Initial With Clamper',sRcyText:='Sensor Timeout Expired Before Operation Completed. Sensor Operation Is Abnormal. Solve The Error To Resume Operation.'),(sAlmText:='Clamper Clamp Safety Sensor Error In Clamp Check While Conveyor Initial With Clamper',sRcyText:='Safety System Has Been Triggered. All Operations Are Disable. Remove the Obstacle That Triggered The Safety Interlock To Resume Operation.'),(sAlmText:='Magazine Not Detected While Pre-Exiting Magazine',sRcyText:='Operation Interrupted By Undetected Magazine. Adjusting The Magazine Or Remove The Present Magazine To Resume Operation.'),(sAlmText:='Magazine Width Check Sensor Deactivated',sRcyText:='Please Check the Magazine Width'),(sAlmText:='Saftey Sensor Is Deactivated To Clamp',sRcyText:='Please Check Safety Sensor'),51(0)];
END_VAR
(**)
(*Local Output*)
VAR
	bHvMag : BOOL := FALSE;
	bMtrSigOnOrLToR : BOOL := FALSE;
	bMtrDirOrRToL : BOOL := FALSE;
	bFixClprClampCtrl : BOOL;
	bRmtClprClampCtrl : BOOL;
	bClprTwoOutputControl : BOOL := FALSE;
END_VAR
(**)
(*Local Input*)
VAR
	udiRstErr : UDINT := 0;
	bPrep : BOOL := TRUE;
	bEn : BOOL := TRUE;
	bDis : BOOL := FALSE;
	bManual : BOOL := FALSE;
	bOnDirMod : BOOL := FALSE;
	diInitTm : DINT := 10000;
	tMtrOffDlyTm : TIME := T#0S;
	diTxInTimeOut : DINT := 10000;
	diTxOutTimeOut : DINT := 10000;
	eDirection : eConvDir := ConvDirLToR;
	bLeftSen : BOOL := FALSE;
	bRightSen : BOOL := FALSE;
	bFixClprClampSen : BOOL := FALSE;
	bFixClprUnclampSen : BOOL := FALSE;
	bFixClprClampSafetySen : BOOL := TRUE;
	bFixClprUnclampSafetySen : BOOL := TRUE;
	bRmtClprClampSen : BOOL := FALSE;
	bRmtClprUnclampSen : BOOL := FALSE;
	bRmtClprClampSafetySen : BOOL := TRUE;
	bRmtClprUnclampSafetySen : BOOL := TRUE;
	bWidthChkPrep : BOOL := TRUE;
	sProgNm : STRING[15] := 'MagConv2Clp';
	tClprClampTO : TIME := T#20s;
	tClprUnclampTO : TIME := T#20s;
	bNtSettingsLoadDone : BOOL := TRUE;
END_VAR
(**)
(*Local*)
VAR
	bRstErr : BOOL;
	udiRstErrOld : UDINT;
	bInitDone : BOOL;
	bInitialDone : BOOL;
	bReachEnd : BOOL;
	usiStep : USINT;
	usiSubStep : USINT;
	eStatOld : eMagConv2ClpAction := MagConv2ClpActIdle;
	fbInit : fbConvSenToSenTm;
	fbEnt : fbConvSenToSen;
	fbPreExit : fbConvSenToSenTm;
	fbExit : fbConvSenToSenOff;
	fbExit1 : fbConvSenToSenOff1;
	fbStop : fbConvMtrOff;
	fbFixClprClampChk : fbPneuExtRetSenExtChk;
	fbFixClprUnclampChk : fbPneuExtRetSenRetChk;
	fbRmtClprClampChk : fbPneuExtRetSenExtChk;
	fbFixClprDly : TON := (PT:=T#1s);
	fbRmtClprUnclampChk : fbPneuExtRetSenRetChk;
	fbClprDlyTm : TON;
	fbSmallLargeSenDlyTm : TON := (PT:=T#1S);
	fbWidthChk : TON := (PT:=T#30s);
	fbLeftSenDelayTm : TON := (PT:=T#1S);
	fbClpExtChkTm : TON := (PT:=T#200ms);
	udiModuleNum : UDINT := 1901;
END_VAR
```

### MagConv2Clp4.var - Change By Project
```iecst
(*2019-10-30*)
(**)
(*Action & State & Status*)
VAR
	p_MagConv2Clp4Stat : UDINT;
	p_MagConv2Clp4Status : UDINT;
	p_MagConv2Clp4StatTxt : UDINT;
END_VAR
(**)
(*Alarm*)
VAR
	p_MagConv2Clp4AlmData : UDINT;
END_VAR
(**)
(*Output*)
VAR
	p_MagConv2Clp4HvMag : UDINT;
	p_MagConv2Clp4MtrSigOnOrLToR : UDINT;
	p_MagConv2Clp4MtrDirOrRToL : UDINT;
	p_MagConv2Clp4FixClprClampCtrl : UDINT;
	p_MagConv2Clp4RmtClprClampCtrl : UDINT;
	p_MagConv2Clp4ClprTwoOutputCtrl : UDINT;
END_VAR
```

### Program Logical/MagConv/MagConv2Clp4 (IEC) - 1.00.0 - NtConv v5.00.0 , NtPneu v5.00.0

#### InputRef.var
```iecst
(*2019-10-30*)
(**)
(*General*)
VAR
	p_eAct : REFERENCE TO eMagConv2ClpAction;
	p_udiRstErr : REFERENCE TO UDINT;
	p_bPrep : REFERENCE TO BOOL;
	p_bEn : REFERENCE TO BOOL;
	p_bDis : REFERENCE TO BOOL;
END_VAR
(**)
(*Configuration*)
VAR
	p_bManual : REFERENCE TO BOOL;
	p_bOnDirMod : REFERENCE TO BOOL;
	p_diInitTm : REFERENCE TO DINT;
	p_tMtrOffDlyTm : REFERENCE TO TIME;
	p_diTxInTimeOut : REFERENCE TO DINT;
	p_diTxOutTimeOut : REFERENCE TO DINT;
	p_eDirection : REFERENCE TO eConvDir;
	p_sProgNm : REFERENCE TO STRING[15];
	p_tClprClampTO : REFERENCE TO TIME;
	p_tClprUnclampTO : REFERENCE TO TIME;
	p_bNtSettingsLoadDone : REFERENCE TO BOOL;
END_VAR
(**)
(*Input*)
VAR
	p_bLeftSen : REFERENCE TO BOOL;
	p_bRightSen : REFERENCE TO BOOL;
	p_bFixClprClampSen : REFERENCE TO BOOL;
	p_bFixClprUnclampSen : REFERENCE TO BOOL;
	p_bRmtClprClampSen : REFERENCE TO BOOL;
	p_bRmtClprUnclampSen : REFERENCE TO BOOL;
	p_bFixClprClampSafetySen : REFERENCE TO BOOL;
	p_bFixClprUnclampSafetySen : REFERENCE TO BOOL;
	p_bRmtClprClampSafetySen : REFERENCE TO BOOL;
	p_bRmtClprUnclampSafetySen : REFERENCE TO BOOL;
END_VAR
```

#### InputRef_Link.var
```iecst
(*2019-10-30*)
(**)
VAR
	p_bLinkOpsRun : REFERENCE TO BOOL;
END_VAR
(**)
VAR
	p_bLinkDISafetyRlySig : REFERENCE TO BOOL;
	p_bLinkMagSmallSen : REFERENCE TO BOOL;
	p_bLinkMagLargeSen : REFERENCE TO BOOL;
	p_bLinkFixClprUnClampSen : REFERENCE TO BOOL;
	p_bLinkFixClprClampSen : REFERENCE TO BOOL;
	p_bLinkMagOpsStepMagMtyExit : REFERENCE TO BOOL;
	p_bLinkDIMagEntSen : REFERENCE TO BOOL;
	p_bLinkDO : REFERENCE TO tyDigitalOutput;
	p_bLinkNtParamMagModelAutoVerify : REFERENCE TO BOOL;
END_VAR
```

#### Local.var
```iecst
(*2019-10-30*)
(**)
(*Local Action, State & Status*)
VAR
	eAct : eMagConv2ClpAction := MagConv2ClpActIdle;
	eStat : eMagConv2ClpAction := MagConv2ClpActIdle;
	eStatus : eFBStatus := Idle;
	udiStatus : UDINT := 0;
	sStatTxt : STRING[200] := '';
	a_sStatText : ARRAY[0..50] OF STRING[200] := ['Idling','Initializing','Initializing With Stop Then Clamper','Initializing With Clamper Then Stop','Entering Board','Entering Board With Stop Then Clamper','Entering Board With Clamper Then Stop','Pre-Exiting Board','Pre-Exiting Board With Clamper',2('Exiting Board'),2('Exiting Board With Clamper'),'Fix/Bottom Clamper Setting All Control','Fix/Bottom Clamper Resetting All Control','Fix/Bottom Clamper Setting Clamp','Fix/Bottom Clamper Setting Unclamp','Fix/Bottom Clamper Clamp','Fix/Bottom Clampler Unclamp','Remote/Top Clamper Setting All Control','Remote/Top Clamper Resetting All Control','Remote/Top Clamper Setting Clamp','Remote/Top Clamper Setting Unclamp','Remote/Top Clamper Clamp','Remote/Top Clampler Unclamp','Stopping','Stopping With Clamper','Turning On Motor Signal','Turning On Motor Direction','Turning Off Motor Signal','Turning Off Motor Direction','Turning On All Motor Output','Turning Off All Motor Output',18('')];
END_VAR
(**)
(*Local Alarm*)
VAR
	tyAlmData : tyAlmDat;
	a_tyAlmText : ARRAY[10000..10099] OF tyAlmTxt := [(sAlmText:='Magazine Detected But Not Present At Outlet Sensor (L - R) While Magazine Conveyor Initial',sRcyText:='Operation Interrupted By Undetected Magazine. Adjusting The Magazine Or Remove The Present Magazine To Resume Operation.'),(sAlmText:='Magazine Detected But Not Present At Outlet Sensor (R - L) While Magazine Conveyor Initial',sRcyText:='Operation Interrupted By Undetected Magazine. Adjusting The Magazine Or Remove The Present Magazine To Resume Operation.'),(sAlmText:='Clamper Clamp Sensor Off Time Out In Unclamp Check While Conveyor Initial With Clamper',sRcyText:='Sensor Timeout Expired Before Operation Completed. Sensor Operation Is Abnormal. Solve The Error To Resume Operation.'),(sAlmText:='Clamper Unclamp Sensor On Time Out In Unclamp Check While Conveyor Initial With Clamper',sRcyText:='Sensor Timeout Expired Before Operation Completed. Sensor Operation Is Abnormal. Solve The Error To Resume Operation.'),(sAlmText:='Clamper Unclamp Safety Sensor Error In Unclamp Check While Conveyor Initial With Clamper',sRcyText:='Safety System Has Been Triggered. All Operations Are Disable. Remove the Obstacle That Triggered The Safety Interlock To Resume Operation.'),(sAlmText:='Magazine Detected But Not Present At Outlet Sensor (L - R) While Conveyor Initial With Clamper',sRcyText:='Operation Interrupted By Undetected Magazine. Adjusting The Magazine Or Remove The Present Magazine To Resume Operation.'),(sAlmText:='Magazine Detected But Not Present At Outlet Sensor (R - L) While Conveyor Initial With Clamper',sRcyText:='Operation Interrupted By Undetected Magazine. Adjusting The Magazine Or Remove The Present Magazine To Resume Operation.'),(sAlmText:='Clamper Clamp Sensor On Time Out In Clamp Check While Conveyor Initial With Clamper',sRcyText:='Sensor Timeout Expired Before Operation Completed. Sensor Operation Is Abnormal. Solve The Error To Resume Operation.'),(sAlmText:='Clamper Unclamp Sensor Off Time Out In Clamp Check While Conveyor Initial With Clamper',sRcyText:='Sensor Timeout Expired Before Operation Completed. Sensor Operation Is Abnormal. Solve The Error To Resume Operation.'),(sAlmText:='Clamper Clamp Safety Sensor Error In Clamp Check While Conveyor Initial With Clamper',sRcyText:='Safety System Has Been Triggered. All Operations Are Disable. Remove the Obstacle That Triggered The Safety Interlock To Resume Operation.'),(sAlmText:='Clamper Clamp Sensor On Time Out In Clamp Check While Conveyor Enter With Clamper',sRcyText:='Sensor Timeout Expired Before Operation Completed. Sensor Operation Is Abnormal. Solve The Error To Resume Operation.'),(sAlmText:='Clamper Unclamp Sensor Off Time Out In Clamp Check While Conveyor Enter With Clamper',sRcyText:='Sensor Timeout Expired Before Operation Completed. Sensor Operation Is Abnormal. Solve The Error To Resume Operation.'),(sAlmText:='Clamper Clamp Safety Sensor Error In Clamp Check While Conveyor Enter With Clamper',sRcyText:='Safety System Has Been Triggered. All Operations Are Disable. Remove the Obstacle That Triggered The Safety Interlock To Resume Operation.'),(sAlmText:='Clamper Clamp Sensor Off Time Out In Unclamp Check While Conveyor Exit With Clamper',sRcyText:='Sensor Timeout Expired Before Operation Completed. Sensor Operation Is Abnormal. Solve The Error To Resume Operation.'),(sAlmText:='Clamper Unclamp Sensor On Time Out In Unclamp Check While Conveyor Exit With Clamper',sRcyText:='Sensor Timeout Expired Before Operation Completed. Sensor Operation Is Abnormal. Solve The Error To Resume Operation.'),(sAlmText:='Clamper Unclamp Safety Sensor Error In Unclamp Check While Conveyor Exit With Clamper',sRcyText:='Safety System Has Been Triggered. All Operations Are Disable. Remove the Obstacle That Triggered The Safety Interlock To Resume Operation.'),(sAlmText:='Clamper Clamp Sensor On Time Out In Clamp Check While Clamper Clamp',sRcyText:='Sensor Timeout Expired Before Operation Completed. Sensor Operation Is Abnormal. Solve The Error To Resume Operation.'),(sAlmText:='Clamper Unclamp Sensor Off Time Out In Clamp Check While Clamper Clamp',sRcyText:='Sensor Timeout Expired Before Operation Completed. Sensor Operation Is Abnormal. Solve The Error To Resume Operation.'),(sAlmText:='Clamper Clamp Safety Sensor Error In Clamp Check While Clamper Clamp',sRcyText:='Safety System Has Been Triggered. All Operations Are Disable. Remove the Obstacle That Triggered The Safety Interlock To Resume Operation.'),(sAlmText:='Clamper Clamp Sensor Off Time Out In Unclamp Check While Clamper Unclamp',sRcyText:='Sensor Timeout Expired Before Operation Completed. Sensor Operation Is Abnormal. Solve The Error To Resume Operation.'),(sAlmText:='Clamper Unclamp Sensor On Time Out In Unclamp Check While Clamper Unclamp',sRcyText:='Sensor Timeout Expired Before Operation Completed. Sensor Operation Is Abnormal. Solve The Error To Resume Operation.'),(sAlmText:='Clamper Unclamp Safety Sensor Error In Unclamp Check While Clamper Unclamp',sRcyText:='Safety System Has Been Triggered. All Operations Are Disable. Remove the Obstacle That Triggered The Safety Interlock To Resume Operation.'),(sAlmText:='Clamper Clamp Sensor Off Time Out In Unclamp Check While Stop With Clamper',sRcyText:='Sensor Timeout Expired Before Operation Completed. Sensor Operation Is Abnormal. Solve The Error To Resume Operation.'),(sAlmText:='Clamper Unclamp Sensor On Time Out In Unclamp Check While Stop With Clamper',sRcyText:='Sensor Timeout Expired Before Operation Completed. Sensor Operation Is Abnormal. Solve The Error To Resume Operation.'),(sAlmText:='Clamper Unclamp Safety Sensor Error In Unclamp Check While Stop With Clamper',sRcyText:='Safety System Has Been Triggered. All Operations Are Disable. Remove the Obstacle That Triggered The Safety Interlock To Resume Operation.'),(sAlmText:='Clamper Clamp Sensor Off Time Out In Unclamp Check While Conveyor Exit With Clamper',sRcyText:='Sensor Timeout Expired Before Operation Completed. Sensor Operation Is Abnormal. Solve The Error To Resume Operation.'),(sAlmText:='Clamper Unclamp Sensor On Time Out In Unclamp Check While Conveyor Exit With Clamper',sRcyText:='Sensor Timeout Expired Before Operation Completed. Sensor Operation Is Abnormal. Solve The Error To Resume Operation.'),(sAlmText:='Clamper Unclamp Safety Sensor Error In Unclamp Check While Conveyor Exit With Clamper',sRcyText:='Safety System Has Been Triggered. All Operations Are Disable. Remove the Obstacle That Triggered The Safety Interlock To Resume Operation.'),2((sAlmText:='Transfer In Time Out While Entering Magazine',sRcyText:='Timeout Expired Before Operation Completed. Transmission Abnormal. Remove the Obstacle (If Exists) To Resume Operation.')),(sAlmText:='Transfer Out Time Out While Exiting Magazine',sRcyText:='Timeout Expired Before Operation Completed. Transmission Abnormal. Remove the Obstacle (If Exists) To Resume Operation.'),(sAlmText:='Transfer Out Time Out While Conveyor Exit With Clamper',sRcyText:='Timeout Expired Before Operation Completed. Transmission Abnormal. Remove the Obstacle (If Exists) To Resume Operation.'),(sAlmText:='Transfer Out Time Out While Exiting Magazine',sRcyText:='Timeout Expired Before Operation Completed. Transmission Abnormal. Remove the Obstacle (If Exists) To Resume Operation.'),(sAlmText:='Transfer Out Time Out While Conveyor Exit With Clamper',sRcyText:='Timeout Expired Before Operation Completed. Transmission Abnormal. Remove the Obstacle (If Exists) To Resume Operation.'),(sAlmText:='Clamper Clamp Sensor On Time Out In Clamp Check While Conveyor Enter With Clamper',sRcyText:='Sensor Timeout Expired Before Operation Completed. Sensor Operation Is Abnormal. Solve The Error To Resume Operation.'),(sAlmText:='Clamper Unclamp Sensor Off Time Out In Clamp Check While Conveyor Enter With Clamper',sRcyText:='Sensor Timeout Expired Before Operation Completed. Sensor Operation Is Abnormal. Solve The Error To Resume Operation.'),(sAlmText:='Clamper Clamp Safety Sensor Error In Clamp Check While Conveyor Enter With Clamper',sRcyText:='Safety System Has Been Triggered. All Operations Are Disable. Remove the Obstacle That Triggered The Safety Interlock To Resume Operation.'),(sAlmText:='Transfer In Time Out While Entering Magazine',sRcyText:='Timeout Expired Before Operation Completed. Transmission Abnormal. Remove the Obstacle (If Exists) To Resume Operation.'),(sAlmText:='Clamper Clamp Sensor Off Time Out In Unclamp Check While Conveyor Initial With Clamper',sRcyText:='Sensor Timeout Expired Before Operation Completed. Sensor Operation Is Abnormal. Solve The Error To Resume Operation.'),(sAlmText:='Clamper Unclamp Sensor On Time Out In Unclamp Check While Conveyor Initial With Clamper',sRcyText:='Sensor Timeout Expired Before Operation Completed. Sensor Operation Is Abnormal. Solve The Error To Resume Operation.'),(sAlmText:='Clamper Unclamp Safety Sensor Error In Unclamp Check While Conveyor Initial With Clamper',sRcyText:='Safety System Has Been Triggered. All Operations Are Disable. Remove the Obstacle That Triggered The Safety Interlock To Resume Operation.'),(sAlmText:='Magazine Detected But Not Present At Outlet Sensor (L - R) While Conveyor Initial With Clamper',sRcyText:='Operation Interrupted By Undetected Magazine. Adjusting The Magazine Or Remove The Present Magazine To Resume Operation.'),(sAlmText:='Magazine Detected But Not Present At Outlet Sensor (R - L) While Conveyor Initial With Clamper',sRcyText:='Operation Interrupted By Undetected Magazine. Adjusting The Magazine Or Remove The Present Magazine To Resume Operation.'),(sAlmText:='Clamper Clamp Sensor On Time Out In Clamp Check While Conveyor Initial With Clamper',sRcyText:='Sensor Timeout Expired Before Operation Completed. Sensor Operation Is Abnormal. Solve The Error To Resume Operation.'),(sAlmText:='Clamper Unclamp Sensor Off Time Out In Clamp Check While Conveyor Initial With Clamper',sRcyText:='Sensor Timeout Expired Before Operation Completed. Sensor Operation Is Abnormal. Solve The Error To Resume Operation.'),(sAlmText:='Clamper Clamp Safety Sensor Error In Clamp Check While Conveyor Initial With Clamper',sRcyText:='Safety System Has Been Triggered. All Operations Are Disable. Remove the Obstacle That Triggered The Safety Interlock To Resume Operation.'),(sAlmText:='Magazine Not Detected While Pre-Exiting Magazine',sRcyText:='Operation Interrupted By Undetected Magazine. Adjusting The Magazine Or Remove The Present Magazine To Resume Operation.'),53(0)];
END_VAR
(**)
(*Local Output*)
VAR
	bHvMag : BOOL := FALSE;
	bMtrSigOnOrLToR : BOOL := FALSE;
	bMtrDirOrRToL : BOOL := FALSE;
	bFixClprClampCtrl : BOOL;
	bRmtClprClampCtrl : BOOL;
	bClprTwoOutputControl : BOOL := FALSE;
END_VAR
(**)
(*Local Input*)
VAR
	udiRstErr : UDINT := 0;
	bPrep : BOOL := TRUE;
	bEn : BOOL := TRUE;
	bDis : BOOL := FALSE;
	bManual : BOOL := FALSE;
	bOnDirMod : BOOL := FALSE;
	diInitTm : DINT := 10000;
	tMtrOffDlyTm : TIME := T#0S;
	diTxInTimeOut : DINT := 10000;
	diTxOutTimeOut : DINT := 10000;
	eDirection : eConvDir := ConvDirLToR;
	bLeftSen : BOOL := FALSE;
	bRightSen : BOOL := FALSE;
	bFixClprClampSen : BOOL := FALSE;
	bFixClprUnclampSen : BOOL := FALSE;
	bFixClprClampSafetySen : BOOL := TRUE;
	bFixClprUnclampSafetySen : BOOL := TRUE;
	bRmtClprClampSen : BOOL := FALSE;
	bRmtClprUnclampSen : BOOL := FALSE;
	bRmtClprClampSafetySen : BOOL := TRUE;
	bRmtClprUnclampSafetySen : BOOL := TRUE;
	sProgNm : STRING[15] := 'MagConv2Clp';
	tClprClampTO : TIME := T#20s;
	tClprUnclampTO : TIME := T#20s;
	bNtSettingsLoadDone : BOOL := TRUE;
END_VAR
(**)
(*Local*)
VAR
	bRstErr : BOOL;
	udiRstErrOld : UDINT;
	bInitDone : BOOL;
	bInitialDone : BOOL;
	bReachEnd : BOOL;
	usiStep : USINT;
	usiSubStep : USINT;
	eStatOld : eMagConv2ClpAction := MagConv2ClpActIdle;
	fbInit : fbConvSenToSenTm;
	fbEnt : fbConvSenToSen;
	fbPreExit : fbConvSenToSenTm;
	fbExit : fbConvSenToSenOff;
	fbExit1 : fbConvSenToSenOff1;
	fbStop : fbConvMtrOff;
	fbFixClprClampChk : fbPneuExtRetSenExtChk;
	fbFixClprUnclampChk : fbPneuExtRetSenRetChk;
	fbRmtClprClampChk : fbPneuExtRetSenExtChk;
	fbRmtClprUnclampChk : fbPneuExtRetSenRetChk;
	fbClprDlyTm : TON;
	fbSmallLargeSenDlyTm : TON := (PT:=T#1S);
	fbLeftSenDelayTm : TON := (PT:=T#1S);
	udiModuleNum : UDINT := 1901;
END_VAR
```

#### Act_Alarm.st
```iecst
(** 2019-10-30 **)
ACTION Act_Alarm:

	//Error
	IF EDGEPOS(eStatus = Error) THEN

		tyAlmData.sProgNm		:= p_sProgNm;
		tyAlmData.udiCode		:= udiStatus;
		tyAlmData.eSeverity		:= AlmSeverityError;
		tyAlmData.udiRunTime	:= tyAlmData.udiRunTime + 1;
		tyAlmData.bAlm			:= TRUE;
		tyAlmData.udiModuleNum  := udiModuleNum;
		g_sMagConv2ClpProgNm		:= p_sProgNm;
		//Get Error Message
		IF tyAlmData.udiCode < 10000 OR tyAlmData.udiCode > 10099 THEN
			tyAlmData.sAlmMsg	:= 'Unknown';
			tyAlmData.sRcyMsg	:= 'Unknown';
		ELSE
			tyAlmData.sAlmMsg	:= a_tyAlmText[tyAlmData.udiCode].sAlmText;
			tyAlmData.sRcyMsg	:= a_tyAlmText[tyAlmData.udiCode].sRcyText;
		END_IF

		sStatTxt	:= tyAlmData.sAlmMsg;

	ELSIF bRstErr AND (tyAlmData.udiCode <> 0) THEN

		tyAlmData.udiCode	:= 0;
		tyAlmData.eSeverity	:= AlmSeverityNA;
		tyAlmData.sAlmMsg	:= '';
		tyAlmData.sRcyMsg	:= '';
		tyAlmData.bAlm			:= FALSE;
		sStatTxt	:= a_sStatText[eStat];

	END_IF

END_ACTION
```

#### Act_InitGlobal.st
```iecst
(** 2019-10-30 **)
ACTION Act_InitGlobal:

	(* Always Change If Project Change *)

	//Pass Data To Link
	p_bLinkOpsRun ACCESS p_OpsRun;

	p_bLinkDISafetyRlySig ACCESS p_DISafetyRlySig;

	p_bLinkMagSmallSen ACCESS p_DIMagConvSmallMagSen4;
	p_bLinkMagLargeSen ACCESS p_DIMagConvLargeMagSen4;
	p_bLinkFixClprUnClampSen ACCESS p_DIMag4FixedUnclampRS;
	p_bLinkFixClprClampSen ACCESS p_DIMag4FixedClampRS;
	p_bLinkDO ACCESS p_DO;
	p_bLinkMagOpsStepMagMtyExit ACCESS p_OpsMagConvLD4MagMtyExit;
	p_bLinkDIMagEntSen ACCESS p_DIMagConvEntSen4;

	p_bLinkNtParamMagModelAutoVerify ACCESS p_NtParamProjMagAutoVerifyPrep;
	//Pass Data To Internal Use
	p_udiRstErr ACCESS p_RstErrReset;
	p_bPrep ACCESS p_NtParamProjMag4ConvPrep;
	p_bManual ACCESS p_UIMnlMod;
	p_bOnDirMod ACCESS p_NtParamMagConv4OnDirMod;
	p_diInitTm ACCESS p_McParamMag4ConvRunTmOut;
	p_tMtrOffDlyTm ACCESS p_NtParamMagConv4MtrOffDlyTm;
	p_diTxInTimeOut ACCESS p_McParamMag4ConvRunTmOut;
	p_diTxOutTimeOut ACCESS p_McParamMag4ConvRunTmOut;
	p_eDirection ACCESS p_NtParamProjMagConvDir;
	p_sProgNm ACCESS p_NtParamMagConv4ProgNm;
	p_tClprClampTO ACCESS p_NtParamMagConv4ClprClampTO;
	p_tClprUnclampTO ACCESS p_NtParamMagConv4ClprUnclampTO;
//	p_bLeftSen ACCESS p_DIMagConvEntSen3;
	p_bRightSen	ACCESS p_DIMagPresentSen4;
//	p_bFixClprClampSen ACCESS p_DIMag3FixedClampRS;
//	p_bFixClprUnclampSen ACCESS p_DIMag3FixedUnclampRS;
//	p_bRmtClprClampSen ACCESS p_DIMag3RemoteClampRS;
//	p_bRmtClprUnclampSen ACCESS p_DIMag3RemoteUnclampRS;
	p_bNtSettingsLoadDone ACCESS p_StartupNtSettingsLoadDone;

	(* Always Change If Project Change *)

END_ACTION
```

#### Act_InitLocal.st
```iecst
(** 2019-10-30 **)
ACTION Act_InitLocal:

	//Input Reference Link To Local Variable
	p_eAct ACCESS ADR(eAct);
	p_udiRstErr ACCESS ADR(udiRstErr);
	p_bPrep ACCESS ADR(bPrep);
	p_bEn ACCESS ADR(bEn);
	p_bDis ACCESS ADR(bDis);

	p_bManual ACCESS ADR(bManual);
	p_bOnDirMod ACCESS ADR(bOnDirMod);
	p_diInitTm ACCESS ADR(diInitTm);
	p_tMtrOffDlyTm ACCESS ADR(tMtrOffDlyTm);
	p_diTxInTimeOut ACCESS ADR(diTxInTimeOut);
	p_diTxOutTimeOut ACCESS ADR(diTxOutTimeOut);
	p_eDirection ACCESS ADR(eDirection);
	p_sProgNm ACCESS ADR(sProgNm);
	p_tClprClampTO ACCESS ADR(tClprClampTO);
	p_tClprUnclampTO ACCESS ADR(tClprUnclampTO);
	p_bNtSettingsLoadDone ACCESS ADR(bNtSettingsLoadDone);
	p_bLeftSen ACCESS ADR(bLeftSen);
	p_bRightSen ACCESS ADR(bRightSen);
	p_bFixClprClampSen ACCESS ADR(bFixClprClampSen);
	p_bFixClprUnclampSen ACCESS ADR(bFixClprUnclampSen);
	p_bFixClprClampSafetySen ACCESS ADR(bFixClprClampSafetySen);
	p_bFixClprUnclampSafetySen ACCESS ADR(bFixClprUnclampSafetySen);
	p_bRmtClprClampSen ACCESS ADR(bRmtClprClampSen);
	p_bRmtClprUnclampSen ACCESS ADR(bRmtClprUnclampSen);
	p_bRmtClprClampSafetySen ACCESS ADR(bRmtClprClampSafetySen);
	p_bRmtClprUnclampSafetySen ACCESS ADR(bRmtClprUnclampSafetySen);

END_ACTION
```

#### Act_Link.st
```iecst
(** 2019-10-30 **)
ACTION Act_Link:

	IF p_bLinkDISafetyRlySig = FALSE THEN
		bFixClprClampCtrl	:= FALSE;
		bRmtClprClampCtrl	:= FALSE;
	END_IF

	p_bFixClprUnclampSen :=  p_bLinkFixClprUnClampSen;

	IF p_bLinkNtParamMagModelAutoVerify THEN
		fbSmallLargeSenDlyTm(IN:= p_bLinkMagSmallSen OR p_bLinkMagLargeSen);
		IF fbSmallLargeSenDlyTm.Q THEN
			p_bFixClprClampSen := TRUE;
		ELSE
			p_bFixClprClampSen := FALSE;
		END_IF
	ELSE
		p_bFixClprClampSen := p_bLinkFixClprClampSen;
	END_IF

	p_bRmtClprClampSen := p_bLinkDO.bMag4RemoteClampCtrl;
	p_bRmtClprUnclampSen := NOT p_bLinkDO.bMag4RemoteClampCtrl;
	//	p_tMtrOffDlyTm	:= T#200ms;

	IF p_bLinkMagOpsStepMagMtyExit THEN
		fbLeftSenDelayTm(IN:= TRUE, PT:= T#5000ms);
		IF fbLeftSenDelayTm.Q THEN
			p_bLeftSen := p_bLinkDIMagEntSen;
		END_IF
	ELSE
		p_bLeftSen := p_bLinkDIMagEntSen;
		fbLeftSenDelayTm(IN:= FALSE);
	END_IF

END_ACTION
```

#### Act_LinkAction.st
```iecst
(** 2019-10-30 **)
ACTION Act_LinkAction:

	IF p_bLinkOpsRun = TRUE THEN
		p_eAct ACCESS p_OpsMagConvLD4MagConv2ClpAct;
	ELSIF p_bManual = TRUE THEN
		p_eAct ACCESS p_UIMagConv2Clp4Act;
	ELSE
		p_eAct ACCESS ADR(eAct);
	END_IF

END_ACTION
```
